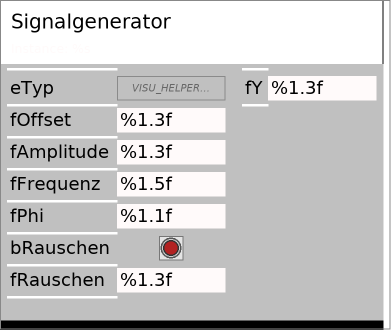
VISUALIZATION RET_VISU_Signalgenerator  // 391x330
VAR_INPUT
   {attribute 'parameterstringof' := 'm_Input_FB'}
   m_Input_INST_Str : STRING;
END_VAR
VAR_IN_OUT
   m_Input_FB : Signalgenerator;
END_VAR
    RoundedRectangle (0,0 383x81)
    RoundedRectangle (0,290 383x40)
    Rectangle (0,64 383x256)
    PushSwitch (159,236 24x24), variable: m_Input_FB.bRauschen, behaviour: TOGGLE, style: Switch-PushSwitch-Red
    Rectangle (8,8 383x27), "Signalgenerator"
    Rectangle (8,35 383x27), "Instance: %s", text variable: m_Input_INST_Str
    Rectangle (7,68 110x2)
    Rectangle (7,76 110x24), "eTyp"
    Rectangle (7,104 110x2)
    Rectangle (117,108 108x24), "%1.3f", text variable: m_Input_FB.fOffset
        OnMouseClick: write the text variable via Default
    Rectangle (7,108 110x24), "fOffset"
    Rectangle (7,136 110x2)
    Rectangle (117,140 108x24), "%1.3f", text variable: m_Input_FB.fAmplitude
        OnMouseClick: write the text variable via Default
    Rectangle (7,140 110x24), "fAmplitude"
    Rectangle (7,168 110x2)
    Rectangle (117,172 108x24), "%1.5f", text variable: m_Input_FB.fFrequenz
        OnMouseClick: write the text variable via Default
    Rectangle (7,172 110x24), "fFrequenz"
    Rectangle (7,200 110x2)
    Rectangle (117,204 108x24), "%1.1f", text variable: m_Input_FB.fPhi
        OnMouseClick: write the text variable via Default
    Rectangle (7,204 110x24), "fPhi"
    Rectangle (7,232 110x2)
    Rectangle (7,236 110x24), "bRauschen"
    Rectangle (7,264 110x2)
    Rectangle (117,268 108x24), "%1.3f", text variable: m_Input_FB.fRauschen
        OnMouseClick: write the text variable via Default
    Rectangle (7,268 110x24), "fRauschen"
    Rectangle (7,296 110x2)
    Rectangle (242,68 26x2)
    Rectangle (268,76 108x24), "%1.3f", text variable: m_Input_FB.fY
    Rectangle (242,76 26x24), "fY"
    Rectangle (242,104 26x2)
    Frame (117,76 108x24), input disabled if: False
        shows VISU_HELPER_Combobox_eSignalform(varEnum := m_Input_FB.eTyp)
END_VISUALIZATION

(* stored: Version 1.1.0.1, ProductVersion 3.1.4024.12
   Visu RET_VISU_Signalgenerator: Id {c7635782-edd2-4f72-a154-137e15a47afd} *)
